FUNCTION_BLOCK FB_Valve
VAR_INPUT
    bEnable        		: BOOL;                 (* Enable valve control *)
    bAuto          		: BOOL;                 (* TRUE = Auto mode, FALSE = Manual mode *)
	b_InOpenFeedback	:BOOL;
	b_InCloseFeedback	:BOOL;	
END_VAR

VAR_OUTPUT
    b_OutOpenCommand   	:  BOOL;  
	b_OutCloseCommand   :  BOOL;       
END_VAR

VAR
	data 		   			: ST_ValveData  ;
	{attribute 'OPC.UA.DA' := '1'}
	{attribute 'OPC.UA.DA.StructuredType' := '1'}
	bManualOpen    			: BOOL;                 (* Manual open command *)
	{attribute 'OPC.UA.DA' := '1'}
	{attribute 'OPC.UA.DA.StructuredType' := '1'}
    bManualClose   			: BOOL;                 (* Manual close command *)
	{attribute 'OPC.UA.DA' := '1'}
	{attribute 'OPC.UA.DA.StructuredType' := '1'}
    bManualReset   			: BOOL;                 (* Manual reset command *)
    ton_MovementTime   		: TON;                	(* Timer for monitor current operation *)
	bStartMovement			: BOOL;
	bOutOpen				: BOOL;
	bOutClose				: BOOL;
END_VAR

VAR PERSISTENT
	stConfig       : ST_ValveConfig;      (* Valve configuration parameters *)
END_VAR

(* Module State logic *)
IF NOT bEnable THEN
    (* Valve is disabled - reset to OFF state *)
	M_PrivateOff();
    RETURN;
ELSIF bAuto THEN 
	data.eModuleState := E_ModuleState.AUTO;
ELSE
	data.eModuleState := E_ModuleState.MANUAL;
	M_PrivateManualMode();
END_IF


(* Main state handling *)
CASE data.eState OF		
    E_ValveState.VALVE_OPENING:

        IF ton_MovementTime.et >= stConfig.tOpenTimeout THEN
            (* Timeout occurred *)
            data.eState:= E_ValveState.VALVE_FAULT;
            data.fault.active := TRUE;
            data.fault.description := 'opening timeout';
        ELSIF b_InOpenFeedback AND stConfig.bEnableOpenFeedback THEN
           	data.eState:= E_ValveState.VALVE_OPEN;
			data.lastOpenTime := ton_MovementTime.PT ;
			bStartMovement := FALSE;
		ELSIF NOT stConfig.bEnableOpenFeedback THEN
			data.eState:= E_ValveState.VALVE_OPEN;
			bStartMovement := FALSE;
        END_IF

	E_ValveState.VALVE_CLOSING:
        IF ton_MovementTime.et >= stConfig.tCloseTimeout THEN
            (* Timeout occurred *)
            data.eState:= E_ValveState.VALVE_FAULT;
            data.fault.active := TRUE;
            data.fault.description := 'closing timeout';
        ELSIF b_InCloseFeedback AND stConfig.bEnableCloseFeedback THEN
           	data.eState:= E_ValveState.VALVE_CLOSED;
			data.lastOpenTime := ton_MovementTime.PT ;
			bStartMovement := FALSE;
		ELSIF NOT stConfig.bEnableOpenFeedback THEN
			data.eState:= E_ValveState.VALVE_CLOSED;
			bStartMovement := FALSE;
        END_IF

    E_ValveState.VALVE_FAULT:
        (* Fault Handling: Manual reset or auto-clear can be added here *)
        (* In this simple example, it remains in fault state until reset manually *)
	

END_CASE;

ton_MovementTime(IN:=bStartMovement, PT:=T#2147483647MS );

METHOD closeAuto : BOOL
IF data.eModuleState = E_ModuleState.AUTO THEN
	M_PrivateCloseValve();
END_IF
END_METHOD

METHOD PRIVATE M_PrivateCloseValve : BOOL
data.eState := E_ValveState.VALVE_CLOSING;
data.lastCloseTime := T#0S;  (* Reset last open time *)
bStartMovement := TRUE;
data.tElapsedTime := T#0S;
bOutOpen := FALSE;
bOutClose:= TRUE;
END_METHOD

METHOD PRIVATE M_PrivateManualMode : BOOL
IF data.eModuleState = E_ModuleState.MANUAL THEN
	IF bManualOpen THEN 
		bManualOpen := FALSE;
		M_PrivateOpenValve();
	ELSIF bManualClose THEN 
		bManualClose := FALSE;
		M_PrivateCloseValve();
	ELSIF bManualReset THEN 
		bManualReset := FALSE;
		M_resetFault();
	END_IF
END_IF
END_METHOD

METHOD PRIVATE M_PrivateOff : BOOL
data.eState := E_ValveState.VALVE_OFF;
data.lastOpenTime := T#0S;  (* Reset last open time *)
data.tElapsedTime := T#0S;
bOutOpen := FALSE;
bOutClose:= FALSE;
M_resetFault();
END_METHOD

METHOD PRIVATE M_PrivateOpenValve : BOOL
data.eState := E_ValveState.VALVE_OPENING;
data.lastOpenTime := T#0S;  (* Reset last open time *)
bStartMovement := TRUE;
data.tElapsedTime := T#0S;
bOutOpen := TRUE;
bOutClose:= FALSE;
END_METHOD

METHOD M_resetFault : BOOL
data.fault.active := FALSE;
data.fault.description := '';
data.eState := E_ValveState.VALVE_OFF;
END_METHOD

METHOD openAuto : BOOL
IF data.eModuleState = E_ModuleState.AUTO THEN
	M_PrivateOpenValve();
END_IF
END_METHOD

END_FUNCTION_BLOCK

(* stored: Version 1.1.0.1, ProductVersion 3.1.4024.13
   POU FB_Valve: Id {223f022c-0a76-49d4-ae57-cf213fa00f1c}, SpecialFunc None
   Method closeAuto: Id {7a89c71d-7369-417e-973f-91421611a6c9}
   Method M_PrivateCloseValve: Id {cba43f05-a8c9-4052-af4c-6a06949011fb}
   Method M_PrivateManualMode: Id {954b5030-3f47-48e9-bff1-d9126bca9554}
   Method M_PrivateOff: Id {1113a748-e2be-4fbc-afb0-6f13b7c83c5e}
   Method M_PrivateOpenValve: Id {8ff9e2ab-a2a3-4bc9-b355-9361890c27fc}
   Method M_resetFault: Id {3622e483-cd75-48fd-9e02-996e5766221e}
   Method openAuto: Id {7bd24405-0748-4670-81ee-17703a7e4e2c} *)
